// TIA Portal V20 export
TYPE "OPC_DestAssign_Ack"
// stored: Namespace ProductionLine
   STRUCT
      AckSeq : Int;
      SourceNode : String[8];
      TotesID : String[10];
      WMSID : String[20];
      Confirmation : String[1];
   END_STRUCT;
END_TYPE
